{attribute 'no_explicit_call' := 'Do not call the body - Stick to OOP'}
FUNCTION_BLOCK FB_EL2595 EXTENDS FB_IlluminationController_Base IMPLEMENTS I_IlluminationSingleOutput_Mode
VAR
	(*DOX Control*)
	bOutput					AT %Q* 	: BOOL;					// Desired State of Output
	bReset					AT %Q*	: BOOL;					// Terminal reset
	
	(*DC Sync*)
	nStartTime 				AT %Q*	: T_DCTIME64;			// Trigger time stamp
	nActivate				AT %Q*	: USINT; 				// 0 -> 3 use new time in terminal
	
	(*DOX Status*)
	bReadyToActivate		AT %I*	: BOOL := FALSE;		// Terminal ready
	bWarning				AT %I*	: BOOL := FALSE;		// Terminal has warning
	bError					AT %I*	: BOOL := FALSE;		// Terminal has error
	
	(*DC Feedback*)
	nDCFeedback				AT %I*  : USINT := 0;			// Feedback of outputchanel
	

	nImpulseLength 			AT %Q* 	: UDINT := 20000;   	// Impulse length of the lighting period [in 1us]
	nTriggerDelay 			AT %Q* 	: UDINT := 10;			// Delay between lighting and camera trigger [in 100ns]

	{attribute 'hide'}
	eState					: E_StateTerminal;				// Current terminal state
	eTriggerSubState		:(SEQ_WirteTime, SEQ_Activate, SEQ_WaitForFeedback, SEQ_Done); //setting the trigger takes several Ethercat cycles
END_VAR

{attribute 'monitoring' := 'call'}
//Module already has a task - already a trigger active
PROPERTY Busy : BOOL
GET
Busy := (THIS^.eState = E_StateTerminal.TRIGGERING);
END_GET
END_PROPERTY

{attribute 'monitoring' := 'call'}
PROPERTY Duration_1us : UDINT
GET
Duration_1us := THIS^.nImpulseLength;
END_GET
SET
THIS^.nImpulseLength := Duration_1us;
END_SET
END_PROPERTY

{attribute 'monitoring' := 'call'}
PROPERTY Operational : BOOL
GET
Operational := (THIS^.eState = E_StateTerminal.READY) OR (THIS^.eState = E_StateTerminal.TRIGGERING);
END_GET
END_PROPERTY

METHOD PUBLIC Reset : HRESULT
VAR_INPUT
END_VAR
IF NOT THIS^.Operational THEN
	THIS^.eState := E_StateTerminal.RESET;
END_IF
END_METHOD

{attribute 'monitoring' := 'call'}
PROPERTY PUBLIC State : E_StateTerminal
GET
State := THIS^.eState;
END_GET
END_PROPERTY

METHOD PUBLIC Trigger : HRESULT
VAR_INPUT
	//The data type T_DCTIME64 represents the distributed clock system time (abbreviated as DC time) as a linear 64-bit integer value. 
	//The time is expressed in nanoseconds since 1/1/2000 UTC. The smallest unit is a nanosecond.
	//F_GetCurDcTickTime64()
	nDCTimeStamp	: T_DCTIME64;
END_VAR
(* Check if the trigger is minimum 3 EtherCat cycles in future *)
IF nDCTimeStamp < THIS^.NextPossibleTriggerTime  THEN
	Trigger := E_FAIL;
	RETURN;
END_IF

(* Check if not in wrong state *)
IF NOT (THIS^.eState = E_StateTerminal.READY) THEN
	Trigger := E_FAIL;
	RETURN;
END_IF




THIS^.nStartTime := nDCTimeStamp;
THIS^.bOutput := TRUE;
THIS^.nActivate := 0;

THIS^.eTriggerSubState := SEQ_WirteTime;
THIS^.eState := E_StateTerminal.TRIGGERING;
Trigger := S_OK;
END_METHOD

METHOD PUBLIC Update : HRESULT
VAR_INST
	fbTimeout : TON;
END_VAR
(* Check for terminal errors *)
IF THIS^.bError AND NOT (THIS^.eState = E_StateTerminal.RESET) THEN 
	THIS^.eState := E_StateTerminal.ERROR;
END_IF

(* Handle terminal state machine *)
CASE THIS^.eState OF
	(* Reset all control variables *)
	E_StateTerminal.RESET:
		THIS^.bReset := TRUE;
		THIS^.eState := E_StateTerminal.RESETING;
		
	(* Reset all control variables *)
	E_StateTerminal.RESETING:
		THIS^.bReset := FALSE;
		THIS^.eState := E_StateTerminal.INIT;	
		
	(* Enable terminal if ready *)
	E_StateTerminal.INIT:			
		IF THIS^.bReadyToActivate THEN
			THIS^.bReset := FALSE;
			THIS^.fbAlarmGeneral.Clear(0, TRUE);
			THIS^.eState := E_StateTerminal.READY;
		END_IF
	
	(* Terminal is ready *)
	E_StateTerminal.READY:
		THIS^.nStartTime := 0;
		THIS^.bOutput := FALSE;
		THIS^.nActivate := 0;

	(* Terminal is triggering *)
	E_StateTerminal.TRIGGERING:
		CASE eTriggerSubState OF
			SEQ_WirteTime:
				//Wirte TimeStamp, Output and Activate=0 in .Trigger()
				//The next commands are allowed only in the next Ethercat cycle
				eTriggerSubState := SEQ_Activate;
				
			SEQ_Activate:
				// Activate new time
				THIS^.nActivate := 3;
				eTriggerSubState := SEQ_WaitForFeedback;
				
			SEQ_WaitForFeedback:
				// Trigger is done and PulsOffTime is done
				IF ((F_GetCurDcTaskTime64()(*100ns*) > THIS^.nStartTime) AND THIS^.bReadyToActivate) THEN
					THIS^.nActivate := 0;
					eTriggerSubState := SEQ_Done;
					//Ready for next Trigger
					THIS^.eState := E_StateTerminal.READY;
				END_IF

			SEQ_Done:
			;
		END_CASE
	
	
	(* Error occured *)	
	E_StateTerminal.ERROR:
		IF NOT THIS^.fbAlarmGeneral.bRaised THEN
			THIS^.fbAlarmGeneral.Raise(0);	
		END_IF
		
		IF (THIS^.fbAlarmGeneral.eConfirmationState = TcEventConfirmationState.Confirmed) THEN
			THIS^.Reset();			
		END_IF			
END_CASE

(* Timeout if an state is to long active *)
fbTimeout.IN := (THIS^.eState = E_StateTerminal.INIT) OR (THIS^.eState = E_StateTerminal.RESETING) OR (THIS^.eState = E_StateTerminal.TRIGGERING);
fbTimeout.PT := T#5S;
fbTimeout();
IF fbTimeout.Q THEN
	THIS^.eState := E_StateTerminal.ERROR;
END_IF
END_METHOD

END_FUNCTION_BLOCK

(* stored: Version 1.1.0.1, ProductVersion 3.1.4024.12
   POU FB_EL2595: Id {815a7e5a-230d-40df-8f77-64f7efcfde1d}, SpecialFunc None
   Property Busy: Id {011661e4-ad5c-4cde-a80e-7b6da8bb24e9}
   Get Get: Id {fff6d4b9-f582-41bf-a35d-2688bd5abe6a}
   Property Duration_1us: Id {e9158780-1de3-448e-8a61-7b1af690333f}
   Get Get: Id {02f5517d-2306-42b8-9655-034ff37da25d}
   Set Set: Id {873113ff-c8b0-4e5c-84aa-9a136028c713}
   Property Operational: Id {02cc84ae-8a6b-4cd9-a9a3-22bca6c0a6a4}
   Get Get: Id {7d06f281-92bd-49ee-99a6-4850dd6da388}
   Method Reset: Id {58c1846a-0a8d-4269-addc-a521503b7c59}
   Property State: Id {ecb4fecd-45fb-4cea-9ee6-46d8bcecdd76}
   Get Get: Id {5a68018b-a251-4aa7-b1d4-89eaa6b6ac8e}
   Method Trigger: Id {334a3bad-68a8-4cb9-83d8-2d1779f5af01}
   Method Update: Id {612f7be6-9d5e-41e2-8748-647edf2ee5b4} *)
